{attribute 'qualified_only'}
{attribute 'strict'}
TYPE  E_WashState :
(
	 IDLE     := 0,
    WASHING  := 1,
    RINSING  := 2,
    SPINNING := 3,
    DONE     := 4,
    ERROR    := 99
);
END_TYPE

(* stored: Version 1.1.0.1, ProductVersion 3.1.4024.16
   DUT E_WashState: Id {311d956f-1bfa-4c7c-8666-ae817009b0c9} *)
